{attribute 'GeneratedUsingTerminal: EK1100-0000-0018'}
{attribute addProperty BoxType "EK1100-0000-0018"}
{attribute addProperty Id "Beckhoff_EL73xxEK1122Beckhoff_EL73xxEK1122_D359B3E92A_0001_EL7332_0000_0016EL7332_615C2CE546A_0002_EL7332_0000_0017EL7332_615C2CE546A_0003_EL7332_0000_0018EL7332_615C2CE546A_0004_EL7332_0000_0019EL7332_615C2CE546A_0005_EL7332_0000_0020EL7332_615C2CE546A_0006_EL7332_0000_0021EL7332_615C2CE546A_0007_EL7332_0000_0022EL7332_615C2CE546A_0008_EL7332_0000_0023EL7332_615C2CE546A_0009_EL7332_0000_0024EL7332_615C2CE546A_0010_EL7342_0000_0016EL7342_2AE9C6B386A_0011_EL7342_0000_0017EL7342_2AE9C6B386A_0012_EL7342_0000_0018EL7342_2AE9C6B386A_0013_EL7342_0000_0019EL7342_2AE9C6B386A_0014_EL7342_0000_0020EL7342_2AE9C6B386A_0015_EL7342_0000_0021EL7342_2AE9C6B386A_0016_EL7342_0000_0022EL7342_2AE9C6B386A_0017_EL7342_0000_0023EL7342_ADEFCF4088A_0018_EL7342_0035_0019EL7342_2AE9C6B386A_0019_EL7342_0035_0020EL7342_2AE9C6B386"}
{attribute addProperty CRC "1028531424"}
{attribute addProperty Size "1278"}
TYPE Beckhoff_EL73xx_3D4E24E0 EXTENDS EK1100_1FC0878B :
STRUCT
	{attribute addProperty Name "Beckhoff EL73xxEK1122"}
	{attribute addProperty PreviousPort "Beckhoff EL73xx : B"}
	Beckhoff_EL73xxEK1122 : Beckhoff_EL73xxEK1122_D359B3E9;
	{attribute addProperty Name "A_0001(EL7332-0000-0016)"}
	{attribute addProperty PreviousPort "Beckhoff EL73xxEK1122 : C"}
	A_0001_EL7332_0000_0016 : EL7332_615C2CE5;
	{attribute addProperty Name "A_0002(EL7332-0000-0017)"}
	{attribute addProperty PreviousPort "A_0001(EL7332-0000-0016) : B"}
	A_0002_EL7332_0000_0017 : EL7332_615C2CE5;
	{attribute addProperty Name "A_0003(EL7332-0000-0018)"}
	{attribute addProperty PreviousPort "A_0002(EL7332-0000-0017) : B"}
	A_0003_EL7332_0000_0018 : EL7332_615C2CE5;
	{attribute addProperty Name "A_0004(EL7332-0000-0019)"}
	{attribute addProperty PreviousPort "A_0003(EL7332-0000-0018) : B"}
	A_0004_EL7332_0000_0019 : EL7332_615C2CE5;
	{attribute addProperty Name "A_0005(EL7332-0000-0020)"}
	{attribute addProperty PreviousPort "A_0004(EL7332-0000-0019) : B"}
	A_0005_EL7332_0000_0020 : EL7332_615C2CE5;
	{attribute addProperty Name "A_0006(EL7332-0000-0021)"}
	{attribute addProperty PreviousPort "A_0005(EL7332-0000-0020) : B"}
	A_0006_EL7332_0000_0021 : EL7332_615C2CE5;
	{attribute addProperty Name "A_0007(EL7332-0000-0022)"}
	{attribute addProperty PreviousPort "A_0006(EL7332-0000-0021) : B"}
	A_0007_EL7332_0000_0022 : EL7332_615C2CE5;
	{attribute addProperty Name "A_0008(EL7332-0000-0023)"}
	{attribute addProperty PreviousPort "A_0007(EL7332-0000-0022) : B"}
	A_0008_EL7332_0000_0023 : EL7332_615C2CE5;
	{attribute addProperty Name "A_0009(EL7332-0000-0024)"}
	{attribute addProperty PreviousPort "A_0008(EL7332-0000-0023) : B"}
	A_0009_EL7332_0000_0024 : EL7332_615C2CE5;
	{attribute addProperty Name "A_0010(EL7342-0000-0016)"}
	{attribute addProperty PreviousPort "A_0009(EL7332-0000-0024) : B"}
	A_0010_EL7342_0000_0016 : EL7342_2AE9C6B3;
	{attribute addProperty Name "A_0011(EL7342-0000-0017)"}
	{attribute addProperty PreviousPort "A_0010(EL7342-0000-0016) : B"}
	A_0011_EL7342_0000_0017 : EL7342_2AE9C6B3;
	{attribute addProperty Name "A_0012(EL7342-0000-0018)"}
	{attribute addProperty PreviousPort "A_0011(EL7342-0000-0017) : B"}
	A_0012_EL7342_0000_0018 : EL7342_2AE9C6B3;
	{attribute addProperty Name "A_0013(EL7342-0000-0019)"}
	{attribute addProperty PreviousPort "A_0012(EL7342-0000-0018) : B"}
	A_0013_EL7342_0000_0019 : EL7342_2AE9C6B3;
	{attribute addProperty Name "A_0014(EL7342-0000-0020)"}
	{attribute addProperty PreviousPort "A_0013(EL7342-0000-0019) : B"}
	A_0014_EL7342_0000_0020 : EL7342_2AE9C6B3;
	{attribute addProperty Name "A_0015(EL7342-0000-0021)"}
	{attribute addProperty PreviousPort "A_0014(EL7342-0000-0020) : B"}
	A_0015_EL7342_0000_0021 : EL7342_2AE9C6B3;
	{attribute addProperty Name "A_0016(EL7342-0000-0022)"}
	{attribute addProperty PreviousPort "A_0015(EL7342-0000-0021) : B"}
	A_0016_EL7342_0000_0022 : EL7342_2AE9C6B3;
	{attribute addProperty Name "A_0017(EL7342-0000-0023)"}
	{attribute addProperty PreviousPort "A_0016(EL7342-0000-0022) : B"}
	A_0017_EL7342_0000_0023 : EL7342_ADEFCF40;
	{attribute addProperty Name "A_0018(EL7342-0035-0019)"}
	{attribute addProperty PreviousPort "A_0017(EL7342-0000-0023) : B"}
	A_0018_EL7342_0035_0019 : EL7342_2AE9C6B3;
	{attribute addProperty Name "A_0019(EL7342-0035-0020)"}
	{attribute addProperty PreviousPort "A_0018(EL7342-0035-0019) : B"}
	A_0019_EL7342_0035_0020 : EL7342_2AE9C6B3;
END_STRUCT
END_TYPE

(* stored: Version 1.2.0.0, ProductVersion 3.1.4024.9
   DUT Beckhoff_EL73xx_3D4E24E0: Id {6ecf931a-4935-4808-807d-dc6b2c8f71e6} *)
